Fanuc KAREL source: ko00141.KL

-- PROVISIONAL review KL for V770-1; original PC SHA256 12141cab01efaadb5dd36e6c510771a02d80d86e9e7cf389fd2f88a6f5a88cd6
-- Incomplete behavior may be omitted. Consult companion uncertainty JSON. Do not deploy.
PROGRAM KO00141
%NOLOCKGROUP
VAR
  R : REAL
  N : INTEGER
-- UNRESOLVED_DECL CFG type=00001c
-- UNRESOLVED_DECL OUT type=000102
BEGIN
  -- UNRESOLVED_PC offsets 5-12; opcodes 9D,23
  -- UNRESOLVED_PC offsets 17-28; opcodes 2E,23
  -- UNRESOLVED_PC offsets 33-43; opcodes 9D,22,A5
  -- UNRESOLVED_PC offsets 48-107; opcodes 27,22,22,22,27,21,64,22,22,22,76,7E,4A
  -- UNRESOLVED_PC offsets 112-116; opcodes 7F
END KO00141
